// TIA Portal V17 export
// export: Created 2024-06-23T21:09:20.2686495Z, ExportSetting WithDefaults, DisplayName Totally Integrated Automation Portal, DisplayVersion V17, DisplayName TIA Portal Openness, DisplayVersion V17, DisplayName TIA Portal Version Control Interface, DisplayVersion V17, DisplayName STEP 7 Professional, DisplayVersion V17, DisplayName STEP 7 Safety, DisplayVersion V17, DisplayName WinCC Professional, DisplayVersion V17
DATA_BLOCK "St0_Per"   // DB55
{ S7_Optimized_Access := 'TRUE' }
VERSION : 0.1
// stored: AutoNumber false, DBAccessibleFromOPCUA true, DBAccessibleFromWebserver true, IsOnlyStoredInLoadMemory false, IsRetainMemResEnabled false, IsWriteProtectedInAS false, MemoryReserve 100
   VAR RETAIN
      HWID : Struct
         _St1_Axe_X : HW_IO := 279;
         _St1_Axe_Y : HW_IO := 281;
         _St1_Prehenseur_Z : HW_IO := 291;
         _St2_Axe_X1 : HW_IO := 293;
         _St2_Axe_X2 : HW_IO := 303;
         _St2_Prehenseur_Z : HW_IO := 305;
         _St3_Axe_X1 : HW_IO := 315;
         _St3_Axe_X2 : HW_IO := 317;
         _St3_Axe_Y : HW_IO := 327;
         "_St3.Axe_Z" : HW_IO := 387;
         _St4_Axe_X1 : HW_IO := 329;
         _St4_Axe_Y1 : HW_IO := 339;
         _St4_Axe_Y2 : HW_IO := 341;
         _St4_Prehenseur_Z2 : HW_IO := 351;
         _St4_Prehenseur_Z3 : HW_IO := 353;
      END_STRUCT;
   END_VAR
BEGIN
END_DATA_BLOCK
